///EL2901 | Potential supply terminal, TwinSAFE, 24 V DC, 10 A
FUNCTION_BLOCK EL2901_v0_00

END_FUNCTION_BLOCK

(* stored: Version 1.1.0.1, ProductVersion 3.1.4022.6
   POU EL2901_v0_00: Id {4fef0973-994c-4c76-aadd-89bd8c2fcf6e}, SpecialFunc None *)
